FUNCTION_BLOCK MqttClient EXTENDS StateMachine
VAR_INPUT
END_VAR
VAR_OUTPUT
	
END_VAR

VAR
	bPublishing : BOOL;
	bPublished : BOOL;
	bSubscribing : BOOL;
	bSubscribed : BOOL;
	
	uiSubscriptionCounter : UINT := 1;
	uiPublicationCounter : UINT := 1;
	
	aAdsSubscriptionStorage : ARRAY[1..cMaxSubscriptions] OF ST_MqttAdsShell;
	aAdsPublicationStorage : ARRAY[1..cMaxSubscriptions] OF ST_MqttAdsShell;
	
	i : UINT;
	
END_VAR

VAR CONSTANT
	cMaxSubscriptions : UINT := 10;
	cMaxPublications : UINT := 10;
END_VAR

METHOD PROTECTED Busy : BOOL
VAR_INPUT
END_VAR
VAR_INST
	eAdsConnectorBusy : E_AdsConnectorBusy;
END_VAR
END_METHOD

METHOD PROTECTED  Error : BOOL
VAR_INPUT
END_VAR
END_METHOD

METHOD getNewMessage : ST_MqttPayload
VAR_INPUT
	index : UINT;
END_VAR
IF index > 0
	AND index <= cMaxSubscriptions 
THEN
	getNewMessage := aAdsSubscriptionStorage[index].stMqttPayload;
END_IF
END_METHOD

METHOD PROTECTED  Idle : BOOL
VAR_INPUT
END_VAR
END_METHOD

METHOD PROTECTED  Init : BOOL
VAR_INPUT
END_VAR
END_METHOD

METHOD isNewMessage : UINT
VAR_INPUT
	sTopic : STRING(8);
END_VAR
VAR
	i : UINT;
END_VAR
FOR i := 1 TO cMaxSubscriptions
DO
	IF aAdsSubscriptionStorage[i].sTopic = sTopic 
		AND_THEN aAdsSubscriptionStorage[i].bNewMessage
	THEN
		isNewMessage := i;
		RETURN;
	END_IF
	
END_FOR
END_METHOD

METHOD PROTECTED  Prepare : BOOL
VAR_INPUT
END_VAR
END_METHOD

METHOD Publish : BOOL //Return true if published
VAR_INPUT
	sTopic : STRING(8);
	stMqttPayload : ST_MqttPayload;
END_VAR
IF  uiPublicationCounter > cMaxPublications
	OR
 	(
		bPublishing = TRUE 
		AND bPublished = FALSE
 	) 
THEN
	RETURN;
ELSIF bPublishing = TRUE
	AND bPublished = TRUE
THEN
	bPublishing := FALSE;
	bPublished := FALSE;
	Publish := TRUE;
	RETURN;
END_IF
	
aAdsPublicationStorage[uiPublicationCounter].stMqttPayload := stMqttPayload;
aAdsPublicationStorage[uiPublicationCounter].sTopic := sTopic;
uiPublicationCounter := uiPublicationCounter + 1;

bPublishing := TRUE;
END_METHOD

METHOD PROTECTED  Ready : BOOL
VAR_INPUT
END_VAR
(*
Check conditions to fire Execute() here and put the StateMachine in Busy mode
*)
END_METHOD

METHOD Subscribe : BOOL  //Return true if subscribed
VAR_INPUT
	sTopic : STRING(8);
	
END_VAR
IF 	uiSubscriptionCounter > cMaxSubscriptions
	OR
 	(
		bSubscribing = TRUE 
		AND bSubscribed = FALSE
 	) 
THEN
	RETURN;
ELSIF bSubscribing = TRUE
	AND bSubscribed = TRUE
THEN
	bSubscribing := FALSE;
	bSubscribed := FALSE;
	Subscribe := TRUE;
	RETURN;
END_IF

aAdsSubscriptionStorage[uiSubscriptionCounter].bPlcInit := TRUE;
aAdsSubscriptionStorage[uiSubscriptionCounter].sTopic := sTopic;
uiSubscriptionCounter := uiSubscriptionCounter + 1;

bSubscribing := TRUE;
END_METHOD

METHOD PROTECTED  Waiting : BOOL
VAR_INPUT
END_VAR
END_METHOD

END_FUNCTION_BLOCK

(* stored: Version 1.1.0.1, ProductVersion 3.1.4024.0
   POU MqttClient: Id {a9904573-1d06-4478-8539-d64d4604b034}, SpecialFunc None
   Folder StateMachine: Id {e219cd41-9610-407f-b4ed-9df13e5fae30}
   Method Busy: Id {fc714c6c-11a3-4bb1-b35e-e4c26c799a3c}
   Method Error: Id {36035d46-88bf-453a-b0c1-0bc62b8a89e5}
   Method getNewMessage: Id {2b8aaccd-97e7-4e22-9aff-94f5dd801ca2}
   Method Idle: Id {f2b37aac-75e1-45d1-adb2-6115990781c2}
   Method Init: Id {6d9582f2-fc30-494a-a725-136ab2304568}
   Method isNewMessage: Id {12c826f3-1d82-472b-9ba8-baf5d56c084c}
   Method Prepare: Id {ac43893e-86e6-4b98-bf1a-bbd127d69842}
   Method Publish: Id {af1bedd9-5057-4118-abdc-a50473914887}
   Method Ready: Id {276525ab-8c0c-4f7e-9451-178516549953}
   Method Subscribe: Id {76f556c2-933e-41ef-8e37-b2f14dd034d4}
   Method Waiting: Id {c489313b-bd3b-4ab8-96a1-8021a3677c8a} *)
